(* CODESYS project NetBaseServicesDemo.2020.2.4.1.project

Project tree, tasks and I/O mapping:
  TCPServerPLC : CODESYS Control Win V3, 3S - Smart Software Solutions GmbH, order no. 305021, version 3.5.11.0
    application ServerApp
      libraries: CAA Segmented Buffer Manager Extern, 3.5.11.0 (CAA Technical Workgroup); CAA Behaviour Model, 3.5.11.0 (CAA Technical Workgroup); Standard, * (System); CAA Net Base Services, 3.5.15.0 (CAA Technical Workgroup); CAA Types Extern, 3.5.13.0 (CAA Technical Workgroup)
      task MainTask (cyclic, interval t#20ms, priority 1) calls PLC_PRG
      function SrvErrorCoder [ST]
      function block Handler [ST]: prvCyclicAction, prvStart, prvResetOutputs, prvAbort
      program Server [CFC]
      program PLC_PRG [ST]
  TCPClientPLC : CODESYS Control Win V3, 3S - Smart Software Solutions GmbH, order no. 305021, version 3.5.11.0
    application ClientApp
      libraries: CAA Segmented Buffer Manager Extern, 3.5.11.0 (CAA Technical Workgroup); Standard, * (System); CAA Net Base Services, 3.5.15.0 (CAA Technical Workgroup); CAA Types Extern, 3.5.13.0 (CAA Technical Workgroup)
      task MainTask (cyclic, interval t#20ms, priority 1) calls PLC_PRG
      function CreateMessage [ST]
      program PLC_PRG [ST]
      program Client [CFC]
  UDPProducerPLC : CODESYS Control Win V3, 3S - Smart Software Solutions GmbH, order no. 305021, version 3.5.11.0
    application ProducerApp
      libraries: CAA Segmented Buffer Manager Extern, 3.5.11.0 (CAA Technical Workgroup); Standard, * (System); CAA Net Base Services, 3.5.15.0 (CAA Technical Workgroup); CAA Types Extern, 3.5.13.0 (CAA Technical Workgroup)
      task MainTask (cyclic, interval t#20ms, priority 1) calls PLC_PRG
      function CreateMessage [ST]
      program PLC_PRG [ST]
      program Producer [CFC]
  UDPConsumerPLC : CODESYS Control Win V3, 3S - Smart Software Solutions GmbH, order no. 305021, version 3.5.11.0
    application ConsumerApp
      libraries: CAA Segmented Buffer Manager Extern, 3.5.11.0 (CAA Technical Workgroup); Standard, * (System); CAA Net Base Services, 3.5.15.0 (CAA Technical Workgroup); CAA Types Extern, 3.5.13.0 (CAA Technical Workgroup)
      task MainTask (cyclic, interval t#20ms, priority 1) calls PLC_PRG
      program Consumer [CFC]
      program PLC_PRG [ST]
*)

// TCPClientPLC/ClientApp/PLC_PRG
PROGRAM PLC_PRG
VAR
END_VAR

Client();

END_PROGRAM

// TCPClientPLC/ClientApp/Client
PROGRAM Client
VAR
	Client : NBS.TCP_Client;
	Write: NBS.TCP_Write;
	Read: NBS.TCP_Read;

	T1: TON;
	TTrig: R_TRIG;
	ATrig: R_TRIG;
	FF: SR;

	sTxData: STRING;
	sRxData: STRING;
	szSize: CAA.SIZE;
    
END_VAR
VAR // added by the converter: edge detectors and wires of the graphical bodies
    _w1, _w2, _w4, _w5 : ANY;
    _w3 : BOOL;
END_VAR

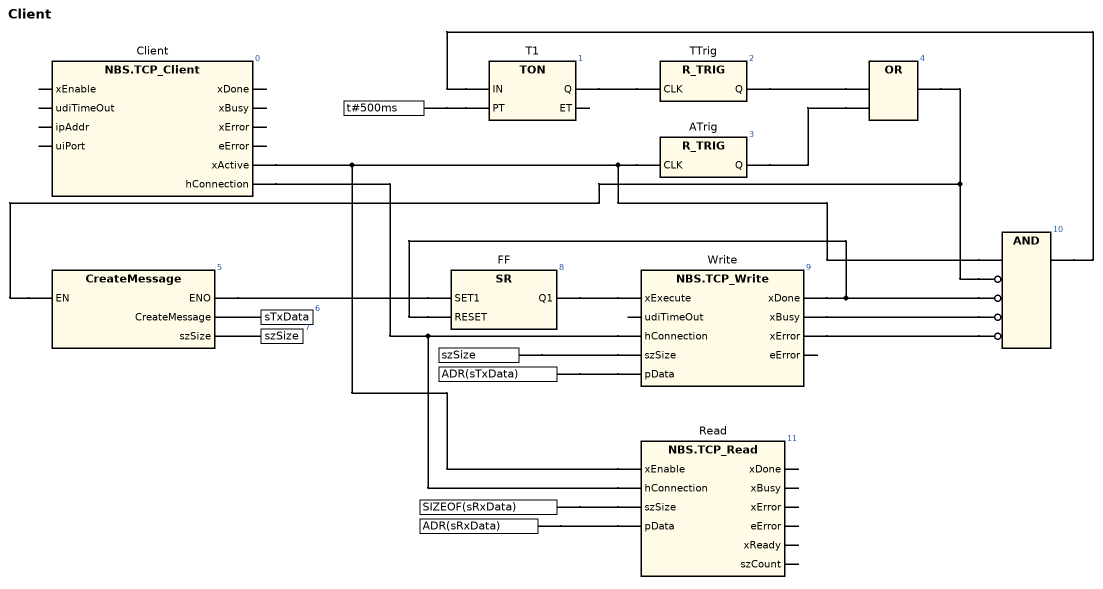
Client(); // NBS.TCP_Client
T1(IN := _w1, PT := t#500ms); // TON
TTrig(CLK := T1.Q); // R_TRIG
ATrig(CLK := Client.xActive); // R_TRIG
_w2 := TTrig.Q OR ATrig.Q;
_w3 := _w2;
IF _w3 THEN _w5 := CreateMessage(szSize => _w4); END_IF
sTxData := _w5;
szSize := _w4;
FF(SET1 := _w3, RESET := Write.xDone); // SR
Write(xExecute := FF.Q1, hConnection := Client.hConnection, szSize := szSize, pData := ADR(sTxData)); // NBS.TCP_Write
_w1 := Client.xActive AND NOT _w2 AND NOT Write.xDone AND NOT Write.xBusy AND NOT Write.xError;
Read(
    xEnable := Client.xActive,
    hConnection := Client.hConnection,
    szSize := SIZEOF(sRxData),
    pData := ADR(sRxData)); // NBS.TCP_Read

END_PROGRAM

// TCPClientPLC/ClientApp/CreateMessage
FUNCTION CreateMessage : STRING
VAR_OUTPUT
	szSize : CAA.SIZE;
END_VAR

CreateMessage := LTIME_TO_STRING(LTIME());
szSize := INT_TO_UINT(LEN(CreateMessage) + 1);

END_FUNCTION

// UDPProducerPLC/ProducerApp/CreateMessage
FUNCTION CreateMessage : STRING
VAR_OUTPUT
	szSize : CAA.SIZE;
END_VAR

CreateMessage := LTIME_TO_STRING(LTIME());
szSize := INT_TO_UINT(LEN(CreateMessage) + 1);

END_FUNCTION

// TCPServerPLC/ServerApp/PLC_PRG
PROGRAM PLC_PRG
VAR
END_VAR

Server();

END_PROGRAM

// TCPServerPLC/ServerApp/Server
PROGRAM Server
VAR
    ipAddr : NBS.IP_ADDR := (sAddr:='0.0.0.0');
	Server: NBS.TCP_Server :=(ipAddr:=ipAddr, uiPort:=8181);
	aHandler : ARRAY[0..2] OF Handler;
END_VAR

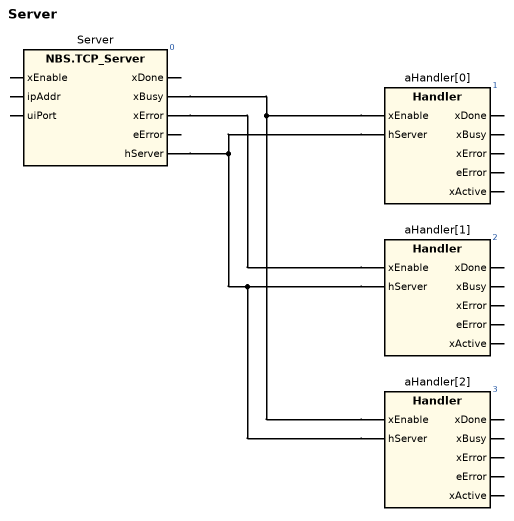
Server(); // NBS.TCP_Server
aHandler[0](xEnable := Server.xBusy, hServer := Server.hServer); // Handler
aHandler[1](xEnable := Server.xError, hServer := Server.hServer); // Handler
aHandler[2](xEnable := Server.xBusy, hServer := Server.hServer); // Handler

END_PROGRAM

// TCPServerPLC/ServerApp/Handler
FUNCTION_BLOCK Handler EXTENDS CBM.LTrig
VAR_INPUT
	hServer : CAA.HANDLE;
END_VAR
VAR_OUTPUT
	eError : NBS.ERROR;
	xActive : BOOL;
END_VAR
VAR
	Con: NBS.TCP_Connection;
	Read : NBS.TCP_ReadBuffer;
	Write : NBS.TCP_WriteBuffer;
	hQueue : CAA.HANDLE;
END_VAR

SUPER^();
eError := iError;

METHOD prvCyclicAction : BOOL
VAR_INPUT
END_VAR
VAR_INST // added by the converter: edge detectors and wires of the graphical bodies
    _w1, _w3, _w4 : ANY;
    _w2 : BOOL;
END_VAR
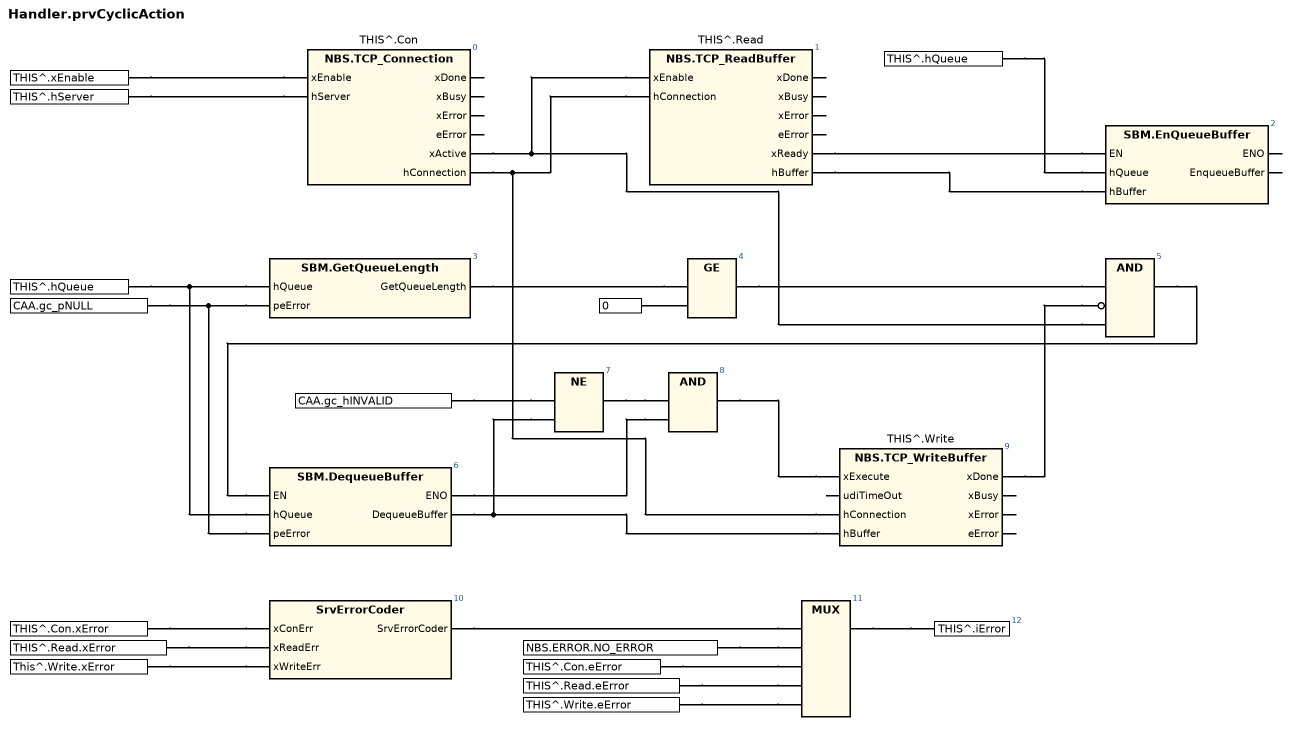
THIS^.Con(xEnable := THIS^.xEnable, hServer := THIS^.hServer); // NBS.TCP_Connection
THIS^.Read(xEnable := THIS^.Con.xActive, hConnection := THIS^.Con.hConnection); // NBS.TCP_ReadBuffer
IF THIS^.Read.xReady THEN SBM.EnQueueBuffer(hQueue := THIS^.hQueue, hBuffer := THIS^.Read.hBuffer); END_IF
_w1 := SBM.GetQueueLength(hQueue := THIS^.hQueue, peError := CAA.gc_pNULL);
_w2 := _w1 >= 0 AND NOT THIS^.Write.xDone AND THIS^.Con.xActive;
IF _w2 THEN _w3 := SBM.DequeueBuffer(hQueue := THIS^.hQueue, peError := CAA.gc_pNULL); END_IF
THIS^.Write(xExecute := CAA.gc_hINVALID <> _w3 AND _w2, hConnection := THIS^.Con.hConnection, hBuffer := _w3); // NBS.TCP_WriteBuffer
_w4 := SrvErrorCoder(xConErr := THIS^.Con.xError, xReadErr := THIS^.Read.xError, xWriteErr := This^.Write.xError);
THIS^.iError := MUX(_w4, NBS.ERROR.NO_ERROR, THIS^.Con.eError, THIS^.Read.eError, THIS^.Write.eError);
END_METHOD

{attribute 'hide'}
METHOD prvStart : BOOL
VAR_INPUT
END_VAR
VAR
END_VAR
THIS^.hQueue := SBM.CreateQueue(peError := ADR(iError));
END_METHOD

{attribute 'hide'}
METHOD prvResetOutputs : BOOL
VAR_INPUT
END_VAR
VAR
END_VAR
(* TODO: insert specific Code here *)
SUPER^.prvResetOutputs();
END_METHOD

{attribute 'hide'}
METHOD prvAbort : BOOL
VAR_INPUT
END_VAR
VAR
END_VAR
IF xError THEN (* abort because of error *)
	(* TODO: insert specific Code here *)
ELSE (* user abort *)
	(* TODO: insert specific Code here *)
END_IF

SBM.DeleteQueue(hQueue := THIS^.hQueue);
hQueue := CAA.gc_hINVALID;

xAbortInProgress:= FALSE;
END_METHOD

END_FUNCTION_BLOCK

// TCPServerPLC/ServerApp/SrvErrorCoder
FUNCTION SrvErrorCoder : INT
VAR_INPUT
	xConErr : BOOL;
	xReadErr : BOOL;
	xWriteErr : BOOL;
END_VAR
VAR
END_VAR

IF xConErr THEN
	SrvErrorCoder := 1;
	RETURN;
END_IF

IF xReadErr THEN
	SrvErrorCoder := 2;
	RETURN;
END_IF

IF xWriteErr THEN
	SrvErrorCoder := 3;
	RETURN;
END_IF

END_FUNCTION

// UDPProducerPLC/ProducerApp/PLC_PRG
PROGRAM PLC_PRG
VAR
END_VAR

Producer();

END_PROGRAM

// UDPProducerPLC/ProducerApp/Producer
PROGRAM Producer
VAR
	Producer : NBS.UDP_Peer;
	Send: NBS.UDP_Send;

	T1: TON;
	TTrig: R_TRIG;
	ATrig: R_TRIG;
	FF: SR;

	sTxData: STRING;
	szSize: CAA.SIZE;
    
END_VAR
VAR // added by the converter: edge detectors and wires of the graphical bodies
    _w1, _w2, _w4, _w5 : ANY;
    _w3 : BOOL;
END_VAR

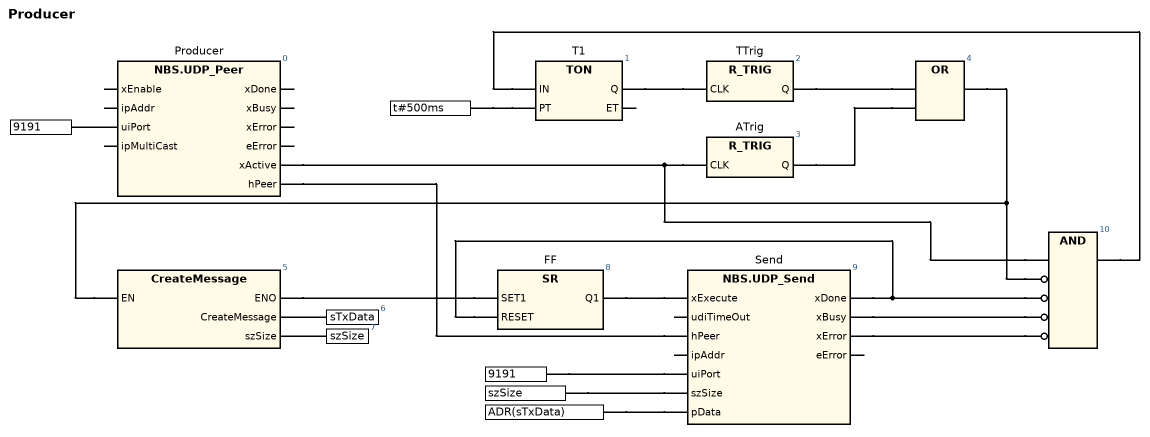
Producer(uiPort := 9191); // NBS.UDP_Peer
T1(IN := _w1, PT := t#500ms); // TON
TTrig(CLK := T1.Q); // R_TRIG
ATrig(CLK := Producer.xActive); // R_TRIG
_w2 := TTrig.Q OR ATrig.Q;
_w3 := _w2;
IF _w3 THEN _w5 := CreateMessage(szSize => _w4); END_IF
sTxData := _w5;
szSize := _w4;
FF(SET1 := _w3, RESET := Send.xDone); // SR
Send(xExecute := FF.Q1, hPeer := Producer.hPeer, uiPort := 9191, szSize := szSize, pData := ADR(sTxData)); // NBS.UDP_Send
_w1 := Producer.xActive AND NOT _w2 AND NOT Send.xDone AND NOT Send.xBusy AND NOT Send.xError;

END_PROGRAM

// UDPConsumerPLC/ConsumerApp/PLC_PRG
PROGRAM PLC_PRG
VAR
END_VAR

Consumer();

END_PROGRAM

// UDPConsumerPLC/ConsumerApp/Consumer
PROGRAM Consumer
VAR
	Consumer : NBS.UDP_Peer;
	Receive: NBS.UDP_ReceiveBuffer;

	sRxData: STRING;
	szSize: CAA.SIZE;
    
    ATrig: R_TRIG;
    BTrig: F_TRIG;
    hQueue : CAA.HANDLE;
END_VAR
VAR // added by the converter: edge detectors and wires of the graphical bodies
    _w1, _w2, _w4, _w6 : ANY;
    _w3, _w5, _w7 : BOOL;
END_VAR

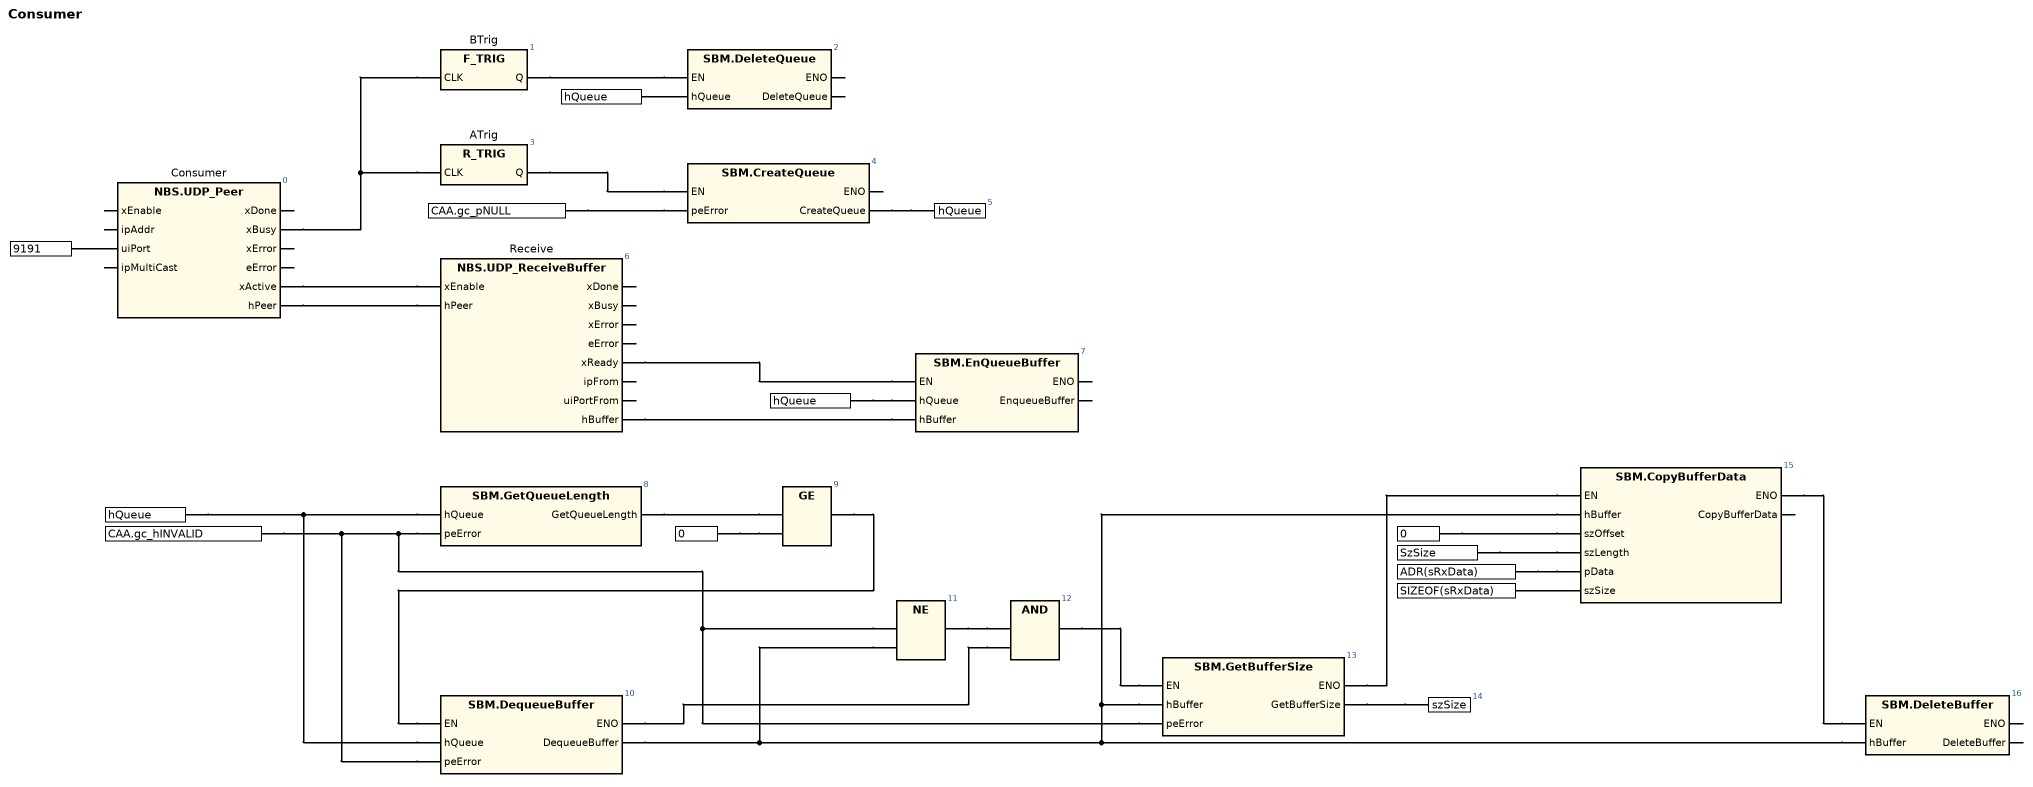
Consumer(uiPort := 9191); // NBS.UDP_Peer
BTrig(CLK := Consumer.xBusy); // F_TRIG
IF BTrig.Q THEN SBM.DeleteQueue(hQueue := hQueue); END_IF
ATrig(CLK := Consumer.xBusy); // R_TRIG
IF ATrig.Q THEN _w1 := SBM.CreateQueue(peError := CAA.gc_pNULL); END_IF
hQueue := _w1;
Receive(xEnable := Consumer.xActive, hPeer := Consumer.hPeer); // NBS.UDP_ReceiveBuffer
IF Receive.xReady THEN SBM.EnQueueBuffer(hQueue := hQueue, hBuffer := Receive.hBuffer); END_IF
_w2 := SBM.GetQueueLength(hQueue := hQueue, peError := CAA.gc_hINVALID);
_w3 := _w2 >= 0;
IF _w3 THEN _w4 := SBM.DequeueBuffer(hQueue := hQueue, peError := CAA.gc_hINVALID); END_IF
_w5 := CAA.gc_hINVALID <> _w4 AND _w3;
IF _w5 THEN _w6 := SBM.GetBufferSize(hBuffer := _w4, peError := CAA.gc_hINVALID); END_IF
szSize := _w6;
_w7 := _w5;
IF _w7 THEN SBM.CopyBufferData(hBuffer := _w4, szOffset := 0, szLength := SzSize, pData := ADR(sRxData), szSize := SIZEOF(sRxData)); END_IF
IF _w7 THEN SBM.DeleteBuffer(hBuffer := _w4); END_IF

END_PROGRAM
